FUNCTION_BLOCK Person_Object EXTENDS TcoCore.TcoObject
VAR
    _RequestedFavor : STRING;
    _ReturnFavor : STRING;
    _refuseFavor : BOOL := FALSE;
    _grantFavor : BOOL := FALSE;
END_VAR

METHOD FavorIsGranted : BOOL
VAR_INPUT
END_VAR
FavorIsGranted := _grantFavor;
END_METHOD

METHOD FavorIsRefused : BOOL
VAR_INPUT
END_VAR
FavorIsRefused := _refuseFavor;
END_METHOD

PROPERTY RequestedFavor : String
GET
RequestedFavor := _RequestedFavor;
END_GET
SET
_RequestedFavor := RequestedFavor;
END_SET
END_PROPERTY

METHOD RequestForTheFavor
VAR_INPUT
    inRequestedFavor : STRING;
    inReturnFavor : STRING;
END_VAR
RequestedFavor := inRequestedFavor;
ReturnFavor := inReturnFavor;
END_METHOD

PROPERTY ReturnFavor : String
GET
ReturnFavor := _ReturnFavor;
END_GET
SET
_ReturnFavor := ReturnFavor;
END_SET
END_PROPERTY

METHOD ThinkCarefully
END_METHOD

END_FUNCTION_BLOCK

(* stored: Version 1.1.0.1, ProductVersion 3.1.4024.6
   POU Person_Object: Id {06d5cb5f-af8e-03ac-15e4-e55d16257585}, SpecialFunc None
   Method FavorIsGranted: Id {ea0055ff-7b27-09bf-256f-625e5bd37bbf}
   Method FavorIsRefused: Id {f98f0004-1b82-0f4d-1c03-f0f82d278e05}
   Property RequestedFavor: Id {180aa208-95eb-07f5-270d-c9f209d9b0ee}
   Get Get: Id {02cea1d1-bba7-0746-19d4-612712dfe3b8}
   Set Set: Id {313bbcfb-1802-06b1-2b48-57d53dcb1bce}
   Method RequestForTheFavor: Id {38491f65-4a1c-0781-37b1-6b079f0ab300}
   Property ReturnFavor: Id {dd89e78c-45ae-034d-1cb3-e75527ef56c0}
   Get Get: Id {ddb5bc1a-2990-0feb-3e5c-16c2e7cd9710}
   Set Set: Id {a4ccb498-833f-0ae2-36b8-f00372fbac57}
   Method ThinkCarefully: Id {920ae051-6065-0815-142d-c6f1b9981c17} *)
